(* IEC 61131-3 sources: MotionTestBenchMaster/Logical/30_MC/Libraries/MotionLib/FC, 11 files *)

(* ---- FC_DegreeToMm.st ---- *)
FUNCTION FC_DegreeToMm
	rTempStep	:= i_rPositionDegree * LREAL_TO_REAL(i_lrMachineStep) / 360.0;

	IF i_xRemindResult THEN
		FC_DegreeToMm	:= FC_RealReminder(i_rDividend := rTempStep, i_rDivisor := LREAL_TO_REAL(i_lrMachineStep), i_rStart := 0);
	ELSE
		FC_DegreeToMm	:= rTempStep;
	END_IF
END_FUNCTION

(* ---- FC_diReminder.st ---- *)
FUNCTION FC_diReminder
	diReminder_a	:= (i_diDividend - (i_diDividend / i_diDivisor) * i_diDivisor);
	diReminder_b	:= (diReminder_a + i_diDivisor - ((diReminder_a + i_diDivisor) / i_diDivisor) * i_diDivisor);

	FC_diReminder	:= (diReminder_b + i_diStart - (((diReminder_b + i_diStart) / i_diDivisor) * i_diDivisor));
END_FUNCTION

(* ---- FC_GetAccFromTimeAndJerk.st ---- *)
(* Get the acceleration (deceleration) value from time and jerk *)
FUNCTION FC_GetAccFromTimeAndJerk
	IF i_rTime = 0 THEN
		rTime := 20;
	ELSE
		rTime := i_rTime;
	END_IF

	IF i_rVelocity <= 0 THEN
		FC_GetAccFromTimeAndJerk :=	500;
		RETURN;
	END_IF

	IF i_rJerk <= 0 THEN
		FC_GetAccFromTimeAndJerk :=	i_rVelocity	/ rTime;
		RETURN;
	ELSE
		rTemp := rTime * rTime - 4 * i_rVelocity / i_rJerk;
		IF rTemp >= 0 THEN
			rTemp := SQRT(rTemp);
			rFistSolution	:= (i_rTime + rTemp) * i_rJerk / 2;
			rSecondSolution	:= (i_rTime - rTemp) * i_rJerk / 2;
			IF i_rVelocity >= (rFistSolution * rFistSolution) / i_rJerk THEN
				FC_GetAccFromTimeAndJerk := rFistSolution;
			ELSIF i_rVelocity >= (rSecondSolution * rSecondSolution) / i_rJerk THEN
				FC_GetAccFromTimeAndJerk := rSecondSolution;
			ELSE
				FC_GetAccFromTimeAndJerk := i_rVelocity / rTime;
			END_IF
		ELSE
			FC_GetAccFromTimeAndJerk :=	i_rVelocity	/ rTime;
		END_IF
	END_IF
END_FUNCTION

(* ---- FC_LongRealReminder.st ---- *)
FUNCTION FC_LongRealReminder
	lrReminder_a	:= (i_lrDividend - (DINT_TO_LREAL(TRUNC(i_lrDividend / i_lrDivisor)) * i_lrDivisor));
	lrReminder_b	:= (lrReminder_a + i_lrDivisor - (DINT_TO_LREAL(TRUNC((lrReminder_a + i_lrDivisor) / i_lrDivisor)) * i_lrDivisor));

	FC_LongRealReminder	:= (lrReminder_b + i_lrStart - (DINT_TO_LREAL(TRUNC((lrReminder_b + i_lrStart) / i_lrDivisor)) * i_lrDivisor));
END_FUNCTION

(* ---- FC_mmToDegree.st ---- *)
FUNCTION FC_mmToDegree
	rTempStep	:= i_rPositionMm * 360.0 / LREAL_TO_REAL(i_lrMachineStep);

	FC_mmToDegree	:= FC_RealReminder(i_rDividend := rTempStep, i_rDivisor := 360.0, i_rStart := 0);
END_FUNCTION

(* ---- FC_RealReminder.st ---- *)
FUNCTION FC_RealReminder
	rReminder_a	:= (i_rDividend - (DINT_TO_REAL(TRUNC(i_rDividend / i_rDivisor)) * i_rDivisor));
	rReminder_b	:= (rReminder_a + i_rDivisor - (DINT_TO_REAL(TRUNC((rReminder_a + i_rDivisor) / i_rDivisor)) * i_rDivisor));

	FC_RealReminder	:= (rReminder_b + i_rStart - (DINT_TO_REAL(TRUNC((rReminder_b + i_rStart) / i_rDivisor)) * i_rDivisor));
END_FUNCTION

(* ---- FC_RephasingMachine.st ---- *)
(* Function for finding the machine rephasing position *)
FUNCTION FC_RephasingMachine
	(* Before starting is necessary to load axes on both arrays *)
	udiLastAxisIndex	:= 0;

	FOR udiAxisIndex := 0 TO 30 BY 1 DO
		alrPositions[udiAxisIndex]	:= 0.0;
		auiAxisIndex[udiAxisIndex]	:= 0;
	END_FOR

	FOR udiAxisIndex := 0 TO CST_LastInletModuleAxis BY 1 DO
		IF iq_astInletSubModuleAxis[udiAxisIndex].iq_stStatus.q_stMainAxisStatus.q_xAxisReal 		AND NOT
			iq_astInletSubModuleAxis[udiAxisIndex].iq_stStatus.q_stMainAxisStatus.q_xPowerSupply 	AND NOT
			iq_astInletSubModuleAxis[udiAxisIndex].iq_stStatus.q_stMainAxisStatus.q_xVelocityControl THEN

			alrPositions[udiLastAxisIndex]	:= iq_astInletSubModuleAxis[udiAxisIndex].iq_stStatus.q_stMainAxisStatus.q_lrPosition;
			auiAxisIndex[udiLastAxisIndex]	:= udiAxisIndex + 2000; (* To the axis module axes index 2000 is added *)

			udiLastAxisIndex	:= MIN(udiLastAxisIndex + 1, 30);
		END_IF
	END_FOR

	FOR udiAxisIndex := 0 TO CST_LastFillerModuleAxis BY 1 DO
		IF iq_astFillerSubModuleAxis[udiAxisIndex].iq_stStatus.q_stMainAxisStatus.q_xAxisReal 		AND NOT
			iq_astFillerSubModuleAxis[udiAxisIndex].iq_stStatus.q_stMainAxisStatus.q_xPowerSupply 	AND NOT
			iq_astFillerSubModuleAxis[udiAxisIndex].iq_stStatus.q_stMainAxisStatus.q_xVelocityControl THEN

			alrPositions[udiLastAxisIndex]	:= iq_astFillerSubModuleAxis[udiAxisIndex].iq_stStatus.q_stMainAxisStatus.q_lrPosition;
			auiAxisIndex[udiLastAxisIndex]	:= udiAxisIndex;

			udiLastAxisIndex	:= MIN(udiLastAxisIndex + 1, 30);
		END_IF
	END_FOR

	FOR udiAxisIndex := 0 TO CST_LastOutletModuleAxis BY 1 DO
		IF iq_astOutletSubModuleAxis[udiAxisIndex].iq_stStatus.q_stMainAxisStatus.q_xAxisReal 			AND NOT
			iq_astOutletSubModuleAxis[udiAxisIndex].iq_stStatus.q_stMainAxisStatus.q_xPowerSupply 		AND NOT
			iq_astOutletSubModuleAxis[udiAxisIndex].iq_stStatus.q_stMainAxisStatus.q_xVelocityControl THEN

			alrPositions[udiLastAxisIndex]	:= iq_astOutletSubModuleAxis[udiAxisIndex].iq_stStatus.q_stMainAxisStatus.q_lrPosition;
			auiAxisIndex[udiLastAxisIndex]	:= udiAxisIndex + 1000; (* To the axis module axes index 1000 is added *)

			udiLastAxisIndex	:= MIN(udiLastAxisIndex + 1, 30);
		END_IF
	END_FOR

	IF udiLastAxisIndex > 1 THEN
		FOR udiRowIndex := 0 TO udiLastAxisIndex - 1 BY 1 DO  (* First Step : make the distance between an axis and the other ones *)
			FOR udiColumnIndex := 0 TO udiLastAxisIndex - 1 BY 1 DO
				aalrDistances[udiRowIndex,udiColumnIndex]	:= 0.0;
				IF udiRowIndex <> udiColumnIndex THEN
					aalrDistances[udiRowIndex,udiColumnIndex] := FC_LongRealReminder(i_lrDividend := (alrPositions[udiRowIndex] - alrPositions[udiColumnIndex]),
					i_lrDivisor:= 360.0,
					i_lrStart:= 0.0);
				END_IF
			END_FOR
		END_FOR

		lrMinimumValue	:= 1e100;
		udiAxisIndex	:= 0;

		FOR udiRowIndex := 0 TO udiLastAxisIndex - 1 BY 1 DO (* Second Step. Verify the path of all axes and find the minimum combination *)
			lrTemp	:= 0;
			FOR udiColumnIndex := 0 TO udiLastAxisIndex - 1 BY 1 DO
				IF udiRowIndex <> udiColumnIndex THEN
					lrTemp := aalrDistances[udiRowIndex, udiColumnIndex]	+ lrTemp;
				END_IF
			END_FOR

			IF lrMinimumValue > lrTemp THEN
				udiAxisIndex		:= udiRowIndex;
				lrMinimumValue		:= lrTemp;
			END_IF
		END_FOR

		FC_RephasingMachine := FC_LongRealReminder(i_lrDividend := alrPositions[udiAxisIndex],
													i_lrDivisor:= 360.0,
													i_lrStart:= 0.0);
	ELSE
		FC_RephasingMachine := FC_LongRealReminder(i_lrDividend:= alrPositions[0],
													i_lrDivisor:= 360.0,
													i_lrStart:= 0.0);
	END_IF
END_FUNCTION

(* ---- FC_RephasingPositionFiller.st ---- *)
(* Find The Position Of The First Axis *)
FUNCTION FC_RephasingPositionFiller
	FOR udiRowIndex := 0 TO CST_LastFillerModuleAxis BY 1 DO (* First Step : make the distance between an axis and the other ones *)
		FOR udiColumnIndex := 0 TO CST_LastFillerModuleAxis BY 1 DO
			aalrDistances[udiRowIndex, udiColumnIndex]	:= 0.0;
			IF 	udiRowIndex <> udiColumnIndex	AND
				iq_astSubModuleAxis[udiRowIndex].iq_stStatus.q_stMainAxisStatus.q_xAxisReal 				AND
				iq_astSubModuleAxis[udiColumnIndex].iq_stStatus.q_stMainAxisStatus.q_xAxisReal 				AND
				NOT iq_astSubModuleAxis[udiRowIndex].iq_stStatus.q_stMainAxisStatus.q_xPowerSupply 			AND
				NOT iq_astSubModuleAxis[udiColumnIndex].iq_stStatus.q_stMainAxisStatus.q_xPowerSupply 		AND
				NOT iq_astSubModuleAxis[udiRowIndex].iq_stStatus.q_stMainAxisStatus.q_xVelocityControl		AND
				NOT iq_astSubModuleAxis[udiColumnIndex].iq_stStatus.q_stMainAxisStatus.q_xVelocityControl THEN

				aalrDistances[udiRowIndex,udiColumnIndex] := FC_LongRealReminder(i_lrDividend := (iq_astSubModuleAxis[udiRowIndex].iq_stStatus.q_stMainAxisStatus.q_lrPosition - iq_astSubModuleAxis[udiColumnIndex].iq_stStatus.q_stMainAxisStatus.q_lrPosition),
																					i_lrDivisor := 360.0,
																					i_lrStart := 0.0);
			END_IF
		END_FOR
	END_FOR

	lrMinimumValue	:= 1e100;
	udiAxisIndex	:= CST_FirstFillerModuleAxis;

	FOR udiRowIndex := 0 TO CST_LastFillerModuleAxis BY 1 DO (* Second Step. Verify the path of all axes and find the minimum combination *)
		lrTemp	:= 0;
		IF iq_astSubModuleAxis[udiRowIndex].iq_stStatus.q_stMainAxisStatus.q_xAxisReal 			AND
			NOT iq_astSubModuleAxis[udiRowIndex].iq_stStatus.q_stMainAxisStatus.q_xPowerSupply 	AND
			NOT iq_astSubModuleAxis[udiRowIndex].iq_stStatus.q_stMainAxisStatus.q_xVelocityControl THEN

			FOR udiColumnIndex := 0 TO CST_LastFillerModuleAxis BY 1 DO
				IF udiRowIndex <> udiColumnIndex AND
					iq_astSubModuleAxis[udiColumnIndex].iq_stStatus.q_stMainAxisStatus.q_xAxisReal  		AND
					NOT iq_astSubModuleAxis[udiColumnIndex].iq_stStatus.q_stMainAxisStatus.q_xPowerSupply 	AND
					NOT iq_astSubModuleAxis[udiColumnIndex].iq_stStatus.q_stMainAxisStatus.q_xVelocityControl THEN

					lrTemp := aalrDistances[udiRowIndex, udiColumnIndex] + lrTemp;
				END_IF
			END_FOR

			IF lrMinimumValue > lrTemp THEN
				udiAxisIndex		:= udiRowIndex;
				lrMinimumValue		:= lrTemp;
			END_IF
		END_IF
	END_FOR

	FC_RephasingPositionFiller := FC_LongRealReminder(i_lrDividend := iq_astSubModuleAxis[udiAxisIndex].iq_stStatus.q_stMainAxisStatus.q_lrPosition,
														i_lrDivisor := 360.0,
														i_lrStart := 0.0);
END_FUNCTION

(* ---- FC_RephasingPositionInlet.st ---- *)
(* Find The Position Of The First Axis *)
FUNCTION FC_RephasingPositionInlet
	FOR udiRowIndex := 0 TO CST_LastInletModuleAxis BY 1 DO (* First Step : make the distance between an axis and the other ones *)
		FOR udiColumnIndex := 0 TO CST_LastInletModuleAxis BY 1 DO
			aalrDistances[udiRowIndex, udiColumnIndex]	:= 0.0;
			IF 	udiRowIndex <> udiColumnIndex	AND
				iq_astSubModuleAxis[udiRowIndex].iq_stStatus.q_stMainAxisStatus.q_xAxisReal 				AND
				iq_astSubModuleAxis[udiColumnIndex].iq_stStatus.q_stMainAxisStatus.q_xAxisReal 				AND
				NOT iq_astSubModuleAxis[udiRowIndex].iq_stStatus.q_stMainAxisStatus.q_xPowerSupply 			AND
				NOT iq_astSubModuleAxis[udiColumnIndex].iq_stStatus.q_stMainAxisStatus.q_xPowerSupply 		AND
				NOT iq_astSubModuleAxis[udiRowIndex].iq_stStatus.q_stMainAxisStatus.q_xVelocityControl		AND
				NOT iq_astSubModuleAxis[udiColumnIndex].iq_stStatus.q_stMainAxisStatus.q_xVelocityControl THEN

				aalrDistances[udiRowIndex,udiColumnIndex] := FC_LongRealReminder(i_lrDividend := (iq_astSubModuleAxis[udiRowIndex].iq_stStatus.q_stMainAxisStatus.q_lrPosition - iq_astSubModuleAxis[udiColumnIndex].iq_stStatus.q_stMainAxisStatus.q_lrPosition),
																				i_lrDivisor := 360.0,
																				i_lrStart := 0.0);
			END_IF
		END_FOR
	END_FOR

	lrMinimumValue	:= 1e100;
	udiAxisIndex	:= CST_FirstInletModuleAxis;

	FOR udiRowIndex := 0 TO CST_LastInletModuleAxis BY 1 DO (* Second Step. Verify the path of all axes and find the minimum combination *)
		lrTemp	:= 0;
		IF iq_astSubModuleAxis[udiRowIndex].iq_stStatus.q_stMainAxisStatus.q_xAxisReal 			AND
			NOT iq_astSubModuleAxis[udiRowIndex].iq_stStatus.q_stMainAxisStatus.q_xPowerSupply 	AND
			NOT iq_astSubModuleAxis[udiRowIndex].iq_stStatus.q_stMainAxisStatus.q_xVelocityControl THEN

			FOR udiColumnIndex := 0 TO CST_LastInletModuleAxis BY 1 DO
				IF udiRowIndex <> udiColumnIndex AND
					iq_astSubModuleAxis[udiColumnIndex].iq_stStatus.q_stMainAxisStatus.q_xAxisReal  		AND
					NOT iq_astSubModuleAxis[udiColumnIndex].iq_stStatus.q_stMainAxisStatus.q_xPowerSupply 	AND
					NOT iq_astSubModuleAxis[udiColumnIndex].iq_stStatus.q_stMainAxisStatus.q_xVelocityControl THEN

					lrTemp := aalrDistances[udiRowIndex, udiColumnIndex] + lrTemp;
				END_IF
			END_FOR

			IF lrMinimumValue > lrTemp THEN
				udiAxisIndex		:= udiRowIndex;
				lrMinimumValue		:= lrTemp;
			END_IF
		END_IF
	END_FOR

	FC_RephasingPositionInlet := FC_LongRealReminder(i_lrDividend := iq_astSubModuleAxis[udiAxisIndex].iq_stStatus.q_stMainAxisStatus.q_lrPosition,
														i_lrDivisor := 360.0,
														i_lrStart := 0.0);
END_FUNCTION

(* ---- FC_RephasingPositionOutlet.st ---- *)
(* Find The Position Of The First Axis *)
FUNCTION FC_RephasingPositionOutlet
	FOR udiRowIndex := 0 TO CST_LastOutletModuleAxis BY 1 DO (* First Step : make the distance between an axis and the other ones *)
		FOR udiColumnIndex := 0 TO CST_LastOutletModuleAxis BY 1 DO
			aalrDistances[udiRowIndex, udiColumnIndex]	:= 0.0;
			IF 	udiRowIndex <> udiColumnIndex	AND
				iq_astSubModuleAxis[udiRowIndex].iq_stStatus.q_stMainAxisStatus.q_xAxisReal 				AND
				iq_astSubModuleAxis[udiColumnIndex].iq_stStatus.q_stMainAxisStatus.q_xAxisReal 				AND
				NOT iq_astSubModuleAxis[udiRowIndex].iq_stStatus.q_stMainAxisStatus.q_xPowerSupply 			AND
				NOT iq_astSubModuleAxis[udiColumnIndex].iq_stStatus.q_stMainAxisStatus.q_xPowerSupply 		AND
				NOT iq_astSubModuleAxis[udiRowIndex].iq_stStatus.q_stMainAxisStatus.q_xVelocityControl		AND
				NOT iq_astSubModuleAxis[udiColumnIndex].iq_stStatus.q_stMainAxisStatus.q_xVelocityControl THEN

				aalrDistances[udiRowIndex,udiColumnIndex] := FC_LongRealReminder(i_lrDividend := (iq_astSubModuleAxis[udiRowIndex].iq_stStatus.q_stMainAxisStatus.q_lrPosition - iq_astSubModuleAxis[udiColumnIndex].iq_stStatus.q_stMainAxisStatus.q_lrPosition),
																					i_lrDivisor := 360.0,
																					i_lrStart := 0.0);
			END_IF
		END_FOR
	END_FOR

	lrMinimumValue	:= 1e100;
	udiAxisIndex	:= CST_FirstOutletModuleAxis;

	FOR udiRowIndex := 0 TO CST_LastOutletModuleAxis BY 1 DO (* Second Step. Verify the path of all axes and find the minimum combination *)
		lrTemp	:= 0;
		IF iq_astSubModuleAxis[udiRowIndex].iq_stStatus.q_stMainAxisStatus.q_xAxisReal 			AND
			NOT iq_astSubModuleAxis[udiRowIndex].iq_stStatus.q_stMainAxisStatus.q_xPowerSupply 	AND
			NOT iq_astSubModuleAxis[udiRowIndex].iq_stStatus.q_stMainAxisStatus.q_xVelocityControl THEN

			FOR udiColumnIndex := 0 TO CST_LastOutletModuleAxis BY 1 DO
				IF udiRowIndex <> udiColumnIndex AND
					iq_astSubModuleAxis[udiColumnIndex].iq_stStatus.q_stMainAxisStatus.q_xAxisReal  		AND
					NOT iq_astSubModuleAxis[udiColumnIndex].iq_stStatus.q_stMainAxisStatus.q_xPowerSupply 	AND
					NOT iq_astSubModuleAxis[udiColumnIndex].iq_stStatus.q_stMainAxisStatus.q_xVelocityControl THEN

					lrTemp := aalrDistances[udiRowIndex, udiColumnIndex] + lrTemp;
				END_IF
			END_FOR

			IF lrMinimumValue > lrTemp THEN
				udiAxisIndex		:= udiRowIndex;
				lrMinimumValue		:= lrTemp;
			END_IF
		END_IF
	END_FOR

	FC_RephasingPositionOutlet := FC_LongRealReminder(i_lrDividend := iq_astSubModuleAxis[udiAxisIndex].iq_stStatus.q_stMainAxisStatus.q_lrPosition,
														i_lrDivisor := 360.0,
														i_lrStart := 0.0);
END_FUNCTION

(* ---- FC_TeensOfmmToDegrees.st ---- *)
FUNCTION FC_TeensOfmmToDegrees
	lrTempStep	:= i_iTeensOfmm * 360.0 / (i_lrMachineStep * 10.0);

	IF i_xWithoutModulo THEN
		FC_TeensOfmmToDegrees := lrTempStep;
	ELSIF i_xNegativeResult THEN
		IF lrTempStep >= 0 THEN
			FC_TeensOfmmToDegrees := FC_LongRealReminder(i_lrDividend := lrTempStep, i_lrDivisor:= 360.0, i_lrStart := 0);
		ELSE
			FC_TeensOfmmToDegrees := FC_LongRealReminder(i_lrDividend := lrTempStep, i_lrDivisor := 360.0, i_lrStart := 0) - 360.0;
		END_IF
	ELSE
		FC_TeensOfmmToDegrees := FC_LongRealReminder(i_lrDividend := lrTempStep, i_lrDivisor := 360.0, i_lrStart:= 0);
	END_IF
END_FUNCTION
